{attribute 'GeneratedUsingTerminal: EK1100-0000-0018'}
{attribute addProperty BoxType "EK1100-0000-0018"}
{attribute addProperty Id "Beckhoff_EL15xxEK1122Beckhoff_EL15xxEK1122_B6563BC52A_0001_EL1502_0000_0000EL1502_3ED4B7F831A_0002_EL1502_0000_0001EL1502_602BA65B32A_0003_EL1502_0000_0016EL1502_602BA65B32A_0004_EL1502_0000_0017EL1502_602BA65B32A_0005_EL1502_0000_0018EL1502_7D732CD532A_0006_EL1502_0000_0019EL1502_7D732CD532A_0007_EL1502_0000_0020EL1502_7D732CD532A_0008_EL1502_0000_0021EL1502_7D732CD532A_0009_EL1502_0000_0022EL1502_7D732CD532A_0010_EL1512_0000_0016EL1512_937D4B1B40A_0011_EL1512_0000_0017EL1512_2F21A4F740A_0012_EL1512_0000_0018EL1512_2F21A4F740A_0013_EL1512_0000_0019EL1512_2F21A4F740A_0014_EL1512_0000_0020EL1512_2F21A4F740A_0015_EL1512_0000_0021EL1512_2F21A4F740"}
{attribute addProperty CRC "3068012975"}
{attribute addProperty Size "529"}
TYPE Beckhoff_EL15xx_B6DE29AF EXTENDS EK1100_AB5A9467 :
STRUCT
	{attribute addProperty Name "Beckhoff_EL15xxEK1122"}
	{attribute addProperty PreviousPort "Beckhoff EL15xx : B"}
	Beckhoff_EL15xxEK1122 : Beckhoff_EL15xxEK1122_B6563BC5;
	{attribute addProperty Name "A_0001_EL1502_0000_0000"}
	{attribute addProperty PreviousPort "Beckhoff EL15xxEK1122 : C"}
	A_0001_EL1502_0000_0000 : EL1502_3ED4B7F8;
	{attribute addProperty Name "A_0002_EL1502_0000_0001"}
	{attribute addProperty PreviousPort "A_0001(EL1502-0000-0000) : B"}
	A_0002_EL1502_0000_0001 : EL1502_602BA65B;
	{attribute addProperty Name "A_0003_EL1502_0000_0016"}
	{attribute addProperty PreviousPort "A_0002(EL1502-0000-0001) : B"}
	A_0003_EL1502_0000_0016 : EL1502_602BA65B;
	{attribute addProperty Name "A_0004_EL1502_0000_0017"}
	{attribute addProperty PreviousPort "A_0003(EL1502-0000-0016) : B"}
	A_0004_EL1502_0000_0017 : EL1502_602BA65B;
	{attribute addProperty Name "A_0005_EL1502_0000_0018"}
	{attribute addProperty PreviousPort "A_0004(EL1502-0000-0017) : B"}
	A_0005_EL1502_0000_0018 : EL1502_7D732CD5;
	{attribute addProperty Name "A_0006_EL1502_0000_0019"}
	{attribute addProperty PreviousPort "A_0005(EL1502-0000-0018) : B"}
	A_0006_EL1502_0000_0019 : EL1502_7D732CD5;
	{attribute addProperty Name "A_0007_EL1502_0000_0020"}
	{attribute addProperty PreviousPort "A_0006(EL1502-0000-0019) : B"}
	A_0007_EL1502_0000_0020 : EL1502_7D732CD5;
	{attribute addProperty Name "A_0008_EL1502_0000_0021"}
	{attribute addProperty PreviousPort "A_0007(EL1502-0000-0020) : B"}
	A_0008_EL1502_0000_0021 : EL1502_7D732CD5;
	{attribute addProperty Name "A_0009_EL1502_0000_0022"}
	{attribute addProperty PreviousPort "A_0008(EL1502-0000-0021) : B"}
	A_0009_EL1502_0000_0022 : EL1502_7D732CD5;
	{attribute addProperty Name "A_0010_EL1512_0000_0016"}
	{attribute addProperty PreviousPort "A_0009(EL1502-0000-0022) : B"}
	A_0010_EL1512_0000_0016 : EL1512_937D4B1B;
	{attribute addProperty Name "A_0011_EL1512_0000_0017"}
	{attribute addProperty PreviousPort "A_0010(EL1512-0000-0016) : B"}
	A_0011_EL1512_0000_0017 : EL1512_2F21A4F7;
	{attribute addProperty Name "A_0012_EL1512_0000_0018"}
	{attribute addProperty PreviousPort "A_0011(EL1512-0000-0017) : B"}
	A_0012_EL1512_0000_0018 : EL1512_2F21A4F7;
	{attribute addProperty Name "A_0013_EL1512_0000_0019"}
	{attribute addProperty PreviousPort "A_0012(EL1512-0000-0018) : B"}
	A_0013_EL1512_0000_0019 : EL1512_2F21A4F7;
	{attribute addProperty Name "A_0014_EL1512_0000_0020"}
	{attribute addProperty PreviousPort "A_0013(EL1512-0000-0019) : B"}
	A_0014_EL1512_0000_0020 : EL1512_2F21A4F7;
	{attribute addProperty Name "A_0015_EL1512_0000_0021"}
	{attribute addProperty PreviousPort "A_0014(EL1512-0000-0020) : B"}
	A_0015_EL1512_0000_0021 : EL1512_2F21A4F7;
END_STRUCT
END_TYPE

(* stored: Version 1.2.0.0, ProductVersion 3.1.4024.9
   DUT Beckhoff_EL15xx_B6DE29AF: Id {8af88542-e35a-4abe-84da-5f034e19a0c7} *)
